INTERFACE I_Navitrol_ReturnToRoute EXTENDS I_Base

METHOD Execute : BOOL
END_METHOD

END_INTERFACE

(* stored: Version 1.1.0.1
   Itf I_Navitrol_ReturnToRoute: Id {c4407225-1f67-420c-9c79-03200eb2cba7}
   Method Execute: Id {1b4d220f-8e03-4f39-999d-fbfa901564cf} *)
